TYPE ST_NovRam_Status :
STRUCT
	nowRowIndex:UDINT;
	writenIndex:UDINT;
	RowDataLocked:ARRAY[0..GVL.NovRamBufferRatio-1]OF BOOL;
	
	
END_STRUCT
END_TYPE

(* stored: Version 1.1.0.1, ProductVersion 3.1.4024.11
   DUT ST_NovRam_Status: Id {117fceb6-7f01-4611-8869-57e3be5a43c8} *)
